Universal Robots PolyScope program: orange_Hospital_base.urp

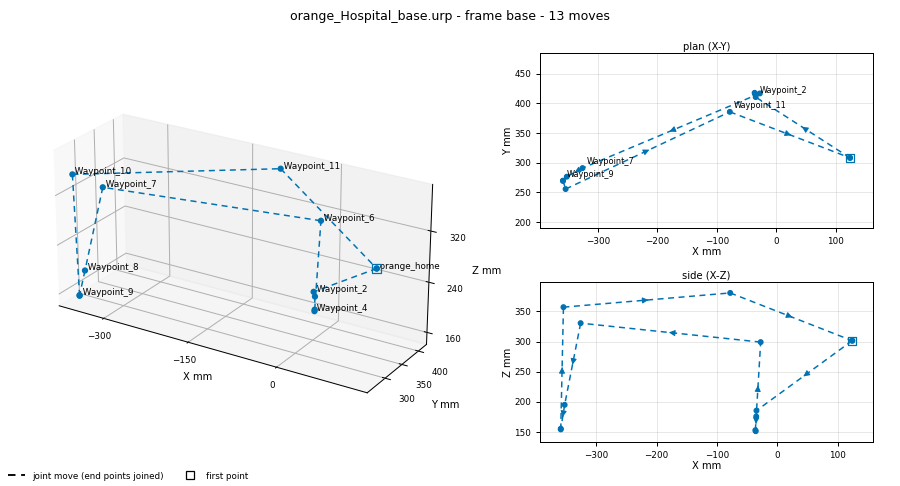
[picture p0: tool path of orange_Hospital_base.urp in frame base, 13 of 13 moves have a stored position in this frame; points joined in program order, loops and branches not executed]
Program orange_Hospital_base (installation=default directory=/programs/usbdisk/Zahra1/orangi createdIn=5.11.11.1010533 lastSavedIn=5.11.11.1010533 robotSerialNumber=20205300864)
Calibrated DH parameters: a=[-0.000166, -0.243494, -0.153108, 0.000057, -0.000123, 0]; d=[0.151897, -1.34267, 53.988124, -52.514559, 0.085283, 0.092193]; alpha=[1.572472, -0.003756, 0.002824, 1.570807, -1.572621, 0]; deltaTheta=[0, 0.020704, 7.033215, -0.770746, 0.000004, 0]
Robot Program (runOnlyOnce=true)
  MoveJ speed 60 deg/s, acceleration 80 deg/s^2 (useActiveTCP=true) feature=Base
    Waypoint orange_home: TCP in base x=124.286 y=308.277 z=301.462 mm, rx=2.2499 ry=-2.1846 rz=-0.0963 rad; joints [-269.66, -91.226, -90.279, -86.086, 92.69, 808.818] deg
    URCap Gripper (Robotiq_Grippers, Robotiq Inc.) dataModel(position=20.0, force=97.0, speed=8.0, positionInDouble=20.0, forceInDouble=97.0, speedInDouble=8.0, slaveIds=[9], blocking=true, robotCompliant=false)
    Waypoint Waypoint_2: TCP in base x=-34.58 y=410.605 z=185.529 mm, rx=2.2362 ry=-2.1606 rz=-0.1449 rad; joints [-247.63, -117.156, -90.107, -58.389, 93.599, 830.684] deg
    Waypoint Waypoint_3: TCP in base x=-34.945 y=415.445 z=175.802 mm, rx=2.2218 ry=-2.15 rz=-0.0693 rad; joints [-247.839, -119.721, -87.48, -61.468, 93.562, 830.465] deg
    Waypoint Waypoint_4: TCP in base x=-35.77 y=416.095 z=151.355 mm, rx=2.2264 ry=-2.1554 rz=-0.0624 rad; joints [-247.663, -122.7, -89.993, -56.047, 93.083, 830.668] deg
    URCap Gripper (Robotiq_Grippers, Robotiq Inc.) dataModel(position=46.666666666666664, force=70.0, speed=56.0, positionInDouble=46.666666666666664, forceInDouble=70.0, speedInDouble=56.0, slaveIds=[9], blocking=true, robotCompliant=false)
    Waypoint Waypoint_5: TCP in base x=-36.372 y=417.751 z=152.975 mm, rx=2.1979 ry=-2.1835 rz=-0.051 rad; joints [-247.642, -122.882, -88.983, -57.241, 92.951, 832.155] deg
    Waypoint Waypoint_6: TCP in base x=-27.581 y=416.739 z=299.112 mm, rx=2.1892 ry=-2.1869 rz=-0.0701 rad; joints [-248.808, -113.787, -62.356, -92.448, 93.411, 831.254] deg
    Waypoint Waypoint_7: TCP in base x=-326.176 y=291.026 z=330.544 mm, rx=-0.0321 ry=-3.0215 rz=-0.0678 rad; joints [-204.433, -117.4, -50.956, -94.253, 90.301, 966.856] deg
    Waypoint Waypoint_8: TCP in base x=-352.67 y=276.519 z=195.064 mm, rx=0.0089 ry=-3.0787 rz=-0.0459 rad; joints [-201.141, -124.069, -75.805, -66.066, 89.636, 968.629] deg
    Waypoint Waypoint_9: TCP in base x=-359.055 y=269.629 z=155.468 mm, rx=-0.0017 ry=-3.1181 rz=-0.1079 rad; joints [-199.34, -128.076, -79.84, -59.505, 86.595, 970.768] deg
    Waypoint Waypoint_12: TCP in base x=-359.123 y=269.655 z=154.31 mm, rx=-0.0016 ry=-3.1182 rz=-0.1078 rad; joints [-199.341, -128.223, -79.925, -59.278, 86.596, 970.763] deg
    URCap Gripper (Robotiq_Grippers, Robotiq Inc.) dataModel(position=1.1764705882352942, force=100.0, speed=100.0, positionInDouble=1.1764705882352942, forceInDouble=100.0, speedInDouble=100.0, slaveIds=[9], blocking=true, robotCompliant=false)
    Waypoint Waypoint_10: TCP in base x=-354.662 y=255.713 z=357.065 mm, rx=-0.0019 ry=-3.1181 rz=-0.1077 rad; joints [-197.607, -123.023, -32.176, -112.317, 86.449, 972.413] deg
    Waypoint Waypoint_11: TCP in base x=-78.105 y=385.721 z=380.645 mm, rx=-1.0924 ry=-2.8926 rz=0.0991 rad; joints [-240.254, -114.138, -38.289, -117.683, 94.453, 971.171] deg
    Waypoint orange_home: TCP in base x=124.286 y=308.277 z=301.462 mm, rx=2.2499 ry=-2.1846 rz=-0.0963 rad; joints [-269.66, -91.226, -90.279, -86.086, 92.69, 808.818] deg
